ORGANIZATION_BLOCK MAIN:OB1
TITLE=New pressure test station
BEGIN
Network 1
	LD     SM0.0
	CALL   PRESSURE_TEST
END_ORGANIZATION_BLOCK
